FUNCTION_BLOCK FB_Cylinder_Sim IMPLEMENTS I_Cylinder
VAR_INPUT
END_VAR
VAR_OUTPUT
END_VAR
VAR
	// original IO
	bAtExtend 		: BOOL;
	bAtRetract 		: BOOL;
	bMoveExtend 	: BOOL;
	bMoveRetract 	: BOOL;
	// internal vars for simulation
	fbTimer				: TON;
	tDelay				: TIME := T#1000MS;
	bStartAtRetractPos	: BOOL := TRUE; // TRUE if default pos is at retract pos
	nState				: INT := 0;
END_VAR

CASE nState OF
	0: // init start position sensor
	IF bStartAtRetractPos THEN
		bAtRetract := TRUE;
	ELSE
		bAtExtend := TRUE;
	END_IF
	nState := nState + 1;
	
	1: // check for move signal
	IF (bMoveExtend AND bAtRetract) THEN
		nState := 10;
	END_IF
	IF (bMoveRetract AND bAtExtend) THEN
		nState := 20;
	END_IF
	
	10: // move to extend pos
	bAtRetract := FALSE;
	fbTimer(IN:=TRUE, PT:=tDelay);
	IF fbTimer.Q THEN
		fbTimer(IN:=FALSE);
		bAtExtend := TRUE;
		nState := 1;
	END_IF
	
	20: // move to retract pos
	bAtExtend := FALSE;
	fbTimer(IN:=TRUE, PT:=tDelay);
	IF fbTimer.Q THEN
		fbTimer(IN:=FALSE);
		bAtRetract := TRUE;
		nState := 1;
	END_IF
	
END_CASE

PROPERTY bIsExtend : BOOL
GET
bIsExtend := bAtExtend;
END_GET
END_PROPERTY

PROPERTY bIsRetract : BOOL
GET
bIsRetract := bAtRetract;
END_GET
END_PROPERTY

METHOD Extend : BOOL
VAR_INPUT
END_VAR
bMoveExtend := TRUE;
bMoveRetract := FALSE;
END_METHOD

METHOD Retract : BOOL
VAR_INPUT
END_VAR
bMoveExtend := FALSE;
bMoveRetract := TRUE;
END_METHOD

END_FUNCTION_BLOCK

(* stored: Version 1.1.0.1, ProductVersion 3.1.4024.12
   POU FB_Cylinder_Sim: Id {ffa2aa7a-79f0-47cd-9215-72e248e615cb}, SpecialFunc None
   Property bIsExtend: Id {d3e10932-1674-48f9-8a46-033d390d7d3b}
   Get Get: Id {1f5dfd04-d882-443f-b16b-33d1d997caf4}
   Property bIsRetract: Id {3ce06607-f8e8-4dac-b4de-bbb6a28b97b6}
   Get Get: Id {d846d01c-b5b3-4ca8-bedb-cb62568d7f9d}
   Method Extend: Id {07f5c472-91d4-46b9-b28b-1968a2e25e39}
   Method Retract: Id {f4d94734-94aa-4b70-92d7-7ee786d9acd5} *)
